(* PLC project , Arduino SRL Arduino PLC IDE Application 1.0.8.0 *)
(* stored: companyURL https://www.axelsoftware.it/, creationDateTime 2026-03-30T20:46:57 *)

VAR_GLOBAL  (* Global_vars *)
  cnt : INT;
END_VAR

VAR_GLOBAL  (* I_O_mappings_ProgInp *)
  BP1 AT %IW0.2 : BOOL;
  BP2 AT %IW0.3 : BOOL;
  BP3 AT %IW0.4 : BOOL;
  BP4 AT %IW0.5 : BOOL;
  PT1 AT %IW0.6 : UINT;
  PT2 AT %IW0.7 : UINT;
  BT1 AT %IW0.0 : BOOL;
  BT2 AT %IW0.1 : BOOL;
END_VAR

VAR_GLOBAL  (* I_O_mappings_RelayOut *)
  LED1 AT %QX0.0 : BOOL;
  LED2 AT %QX0.1 : BOOL;
  LED3 AT %QX0.2 : BOOL;
  LED4 AT %QX0.3 : BOOL;
END_VAR

VAR_GLOBAL  (* I_O_mappings_LEDOut *)
  L1 AT %QX1.0 : BOOL;
  LR AT %QX1.4 : BOOL;
END_VAR

PROGRAM main

cnt := cnt + 1;
END_PROGRAM

CONFIGURATION Configuration
  RESOURCE Resource ON PLC
    VAR_GLOBAL  (* Global_vars *)
      cnt : INT;
    END_VAR
    VAR_GLOBAL  (* I_O_mappings_ProgInp *)
      BP1 AT %IW0.2 : BOOL;
      BP2 AT %IW0.3 : BOOL;
      BP3 AT %IW0.4 : BOOL;
      BP4 AT %IW0.5 : BOOL;
      PT1 AT %IW0.6 : UINT;
      PT2 AT %IW0.7 : UINT;
      BT1 AT %IW0.0 : BOOL;
      BT2 AT %IW0.1 : BOOL;
    END_VAR
    VAR_GLOBAL  (* I_O_mappings_RelayOut *)
      LED1 AT %QX0.0 : BOOL;
      LED2 AT %QX0.1 : BOOL;
      LED3 AT %QX0.2 : BOOL;
      LED4 AT %QX0.3 : BOOL;
    END_VAR
    VAR_GLOBAL  (* I_O_mappings_LEDOut *)
      L1 AT %QX1.0 : BOOL;
      LR AT %QX1.4 : BOOL;
    END_VAR
  END_RESOURCE
END_CONFIGURATION
